TYPE ST_KinematicInfo :
STRUCT
	// Kinematic Info (Value 5)
	KinematicInfo: ARRAY [1..225] OF BYTE;

END_STRUCT
END_TYPE

(* stored: Version 1.1.0.1, ProductVersion 3.1.4020.12
   DUT ST_KinematicInfo: Id {bc1b8b65-5463-4341-9f02-ae2c71841455} *)
